% RSLogix 500 project PLC_TO_TURTLEBOT3.RSS, saved by version 12.00.00.00 %
PROJECT "ML1400"    % processor: MicroLogix 1400 %

PROGRAM FILES
  LAD 2   4 rungs
  LAD 3 "HMI"  5 rungs  % HMI Routine %
  LAD 4 "TELEOP"  7 rungs  % Modbus Routine %
  LAD 5 "COMMAND"  8 rungs

DATA FILES
  O0 OUTPUT  6 elements
  I1 INPUT  8 elements
  S2 STATUS  66 elements
  B3 BINARY  32 elements
  T4 TIMER  1 elements
  C5 COUNTER  1 elements
  R6 CONTROL  1 elements
  N7 INTEGER  20 elements
  F8 FLOAT  10 elements
  N9 HOLD_REG  25 elements
  F10 DECIMALES  7 elements
  N11   6 elements

LADDER 2
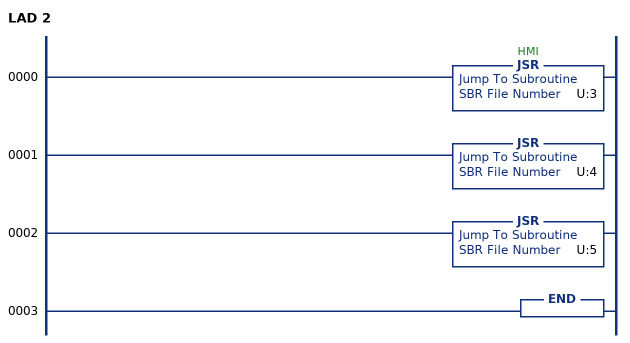
% Rung: 0 %
SOR JSR U:3 EOR
%   U:3  HMI %
% Rung: 1 %
SOR JSR U:4 EOR
% Rung: 2 %
SOR JSR U:5 EOR
% Rung: 3 %
SOR END EOR

LADDER 3 "HMI"    % HMI Routine %
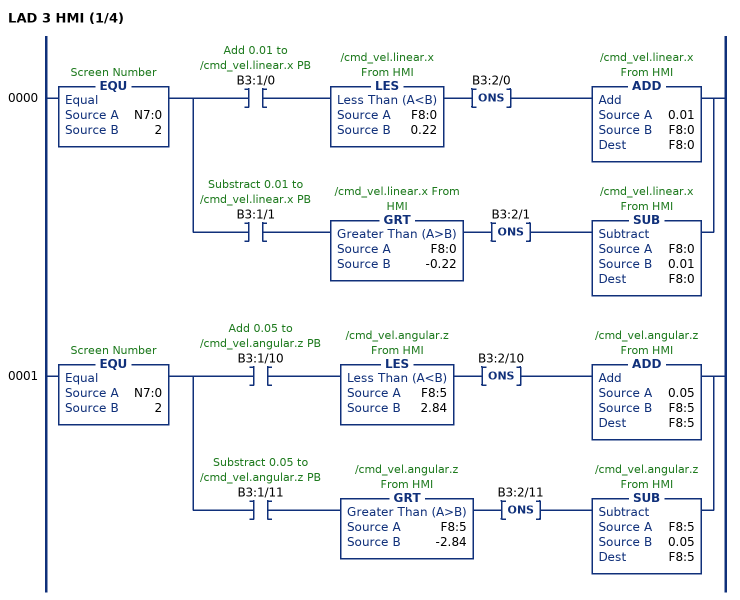
% Rung: 0 %
SOR EQU N7:0 2 BST XIC B3:1/0 LES F8:0 0.22 ONS B3:2/0 ADD 0.01 F8:0 F8:0 NXB XIC B3:1/1 GRT F8:0 -0.22 ONS B3:2/1 SUB F8:0 0.01 F8:0 BND EOR
%   N7:0  "Screen Number" %
%   B3:1/0  "Add 0.01 to /cmd_vel.linear.x PB" %
%   F8:0  "/cmd_vel.linear.x From HMI" %
%   B3:1/1  "Substract 0.01 to /cmd_vel.linear.x PB" %
% Rung: 1 %
SOR EQU N7:0 2 BST XIC B3:1/10 LES F8:5 2.84 ONS B3:2/10 ADD 0.05 F8:5 F8:5 NXB XIC B3:1/11 GRT F8:5 -2.84 ONS B3:2/11 SUB F8:5 0.05 F8:5 BND EOR
%   N7:0  "Screen Number" %
%   B3:1/10  "Add 0.05 to /cmd_vel.angular.z PB" %
%   F8:5  "/cmd_vel.angular.z From HMI" %
%   B3:1/11  "Substract 0.05 to /cmd_vel.angular.z PB" %

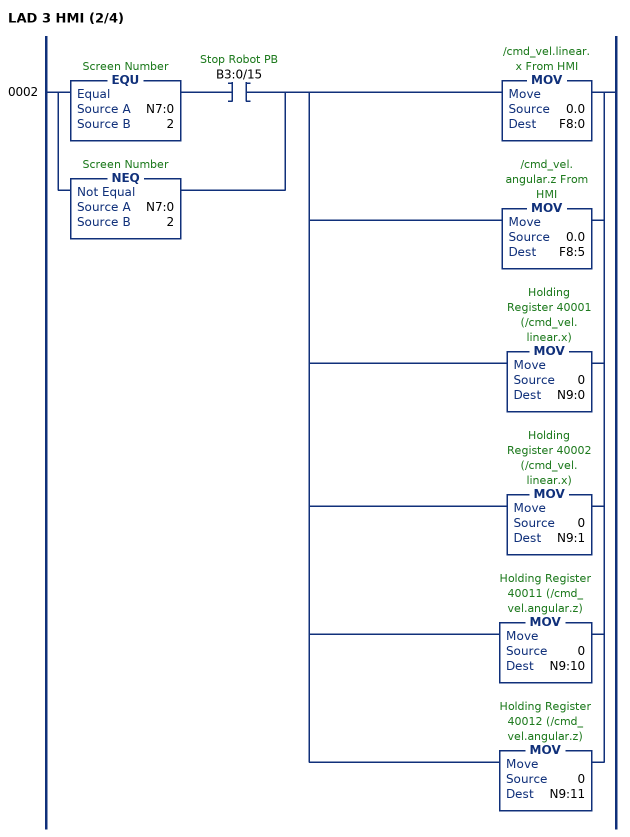
% Rung: 2 %
SOR BST EQU N7:0 2 XIC B3:0/15 NXB NEQ N7:0 2 BND BST MOV 0.0 F8:0 NXB MOV 0.0 F8:5 NXB MOV 0 N9:0 NXB MOV 0 N9:1 NXB MOV 0 N9:10 NXB MOV 0 N9:11 BND EOR
%   N7:0  "Screen Number" %
%   B3:0/15  "Stop Robot PB" %
%   F8:0  "/cmd_vel.linear.x From HMI" %
%   F8:5  "/cmd_vel.angular.z From HMI" %
%   N9:0  "Holding Register 40001 (/cmd_vel.linear.x)" %
%   N9:1  "Holding Register 40002 (/cmd_vel.linear.x)" %
%   N9:10  "Holding Register 40011 (/cmd_vel.angular.z)" %
%   N9:11  "Holding Register 40012 (/cmd_vel.angular.z)" %

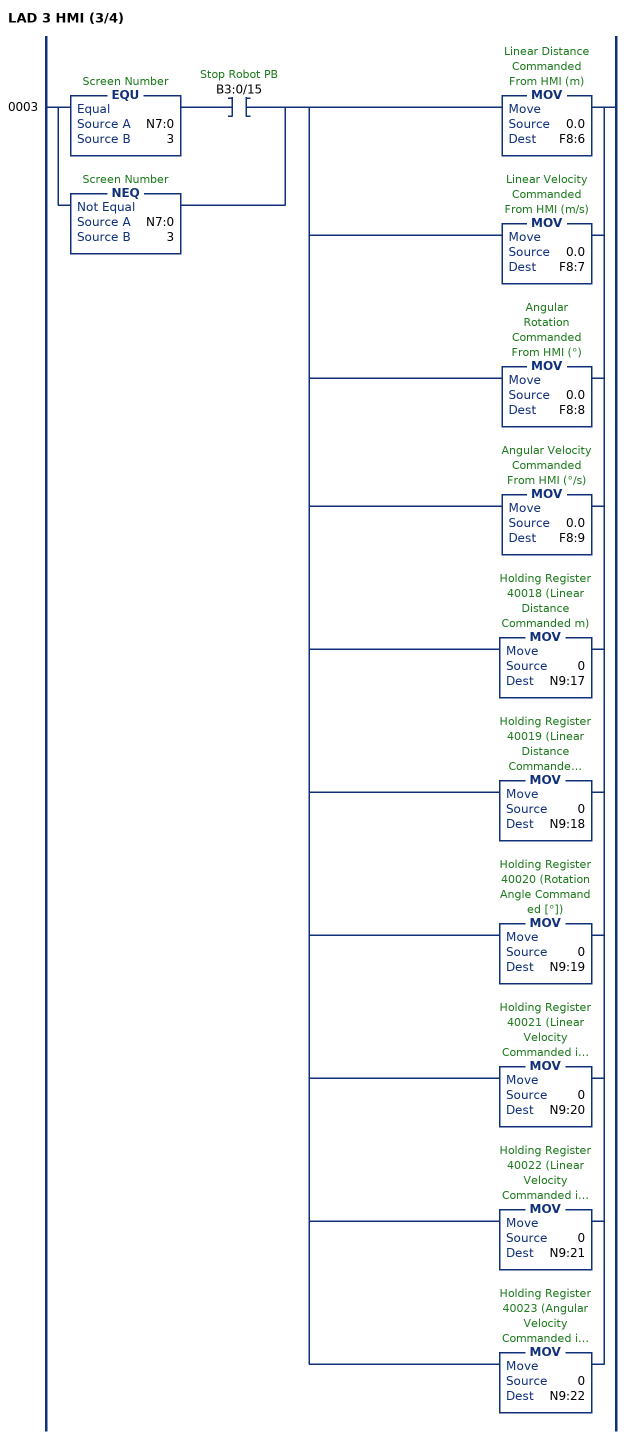
% Rung: 3 %
SOR BST EQU N7:0 3 XIC B3:0/15 NXB NEQ N7:0 3 BND BST MOV 0.0 F8:6 NXB MOV 0.0 F8:7 NXB MOV 0.0 F8:8 NXB MOV 0.0 F8:9 NXB MOV 0 N9:17 NXB MOV 0 N9:18 NXB MOV 0 N9:19 NXB MOV 0 N9:20 NXB MOV 0 N9:21 NXB MOV 0 N9:22 BND EOR
%   N7:0  "Screen Number" %
%   B3:0/15  "Stop Robot PB" %
%   F8:6  "Linear Distance Commanded From HMI (m)" %
%   F8:7  "Linear Velocity Commanded From HMI (m/s)" %
%   F8:8  "Angular Rotation Commanded From HMI (°)" %
%   F8:9  "Angular Velocity Commanded From HMI (°/s)" %
%   N9:17  "Holding Register 40018 (Linear Distance Commanded m)" %
%   N9:18  "Holding Register 40019 (Linear Distance Commanded cm)" %
%   N9:19  "Holding Register 40020 (Rotation Angle Commanded [°])" %
%   N9:20  "Holding Register 40021 (Linear Velocity Commanded in X axis [m])" %
%   N9:21  "Holding Register 40022 (Linear Velocity Commanded in X axis [cm])" %
%   N9:22  "Holding Register 40023 (Angular Velocity Commanded in Z axis [°/s])" %

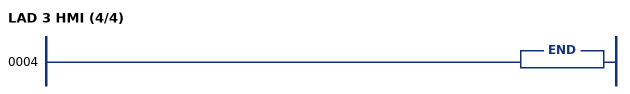
% Rung: 4 %
SOR END EOR

LADDER 4 "TELEOP"    % Modbus Routine %
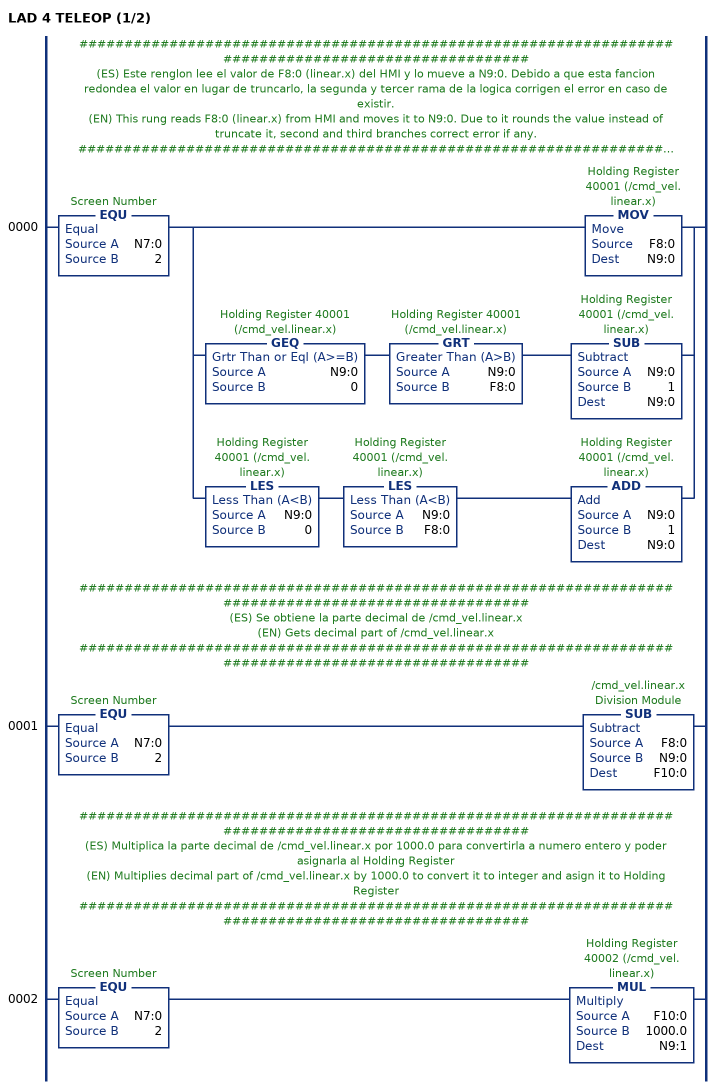
% Rung: 0 %
% ####################################################################################################
% 
% (ES) Este renglon lee el valor de F8:0 (linear.x) del HMI y lo mueve a N9:0. Debido a que esta fancion redondea el valor en lugar de truncarlo, la segunda y tercer rama de la logica corrigen el error en caso de existir.
% (EN) This rung reads F8:0 (linear.x) from HMI and moves it to N9:0. Due to it rounds the value instead of truncate it, second and third branches correct error if any.
% 
% #################################################################################################### %
SOR EQU N7:0 2 BST MOV F8:0 N9:0 NXB GEQ N9:0 0 GRT N9:0 F8:0 SUB N9:0 1 N9:0 NXB LES N9:0 0 LES N9:0 F8:0 ADD N9:0 1 N9:0 BND EOR
%   N7:0  "Screen Number" %
%   F8:0  "/cmd_vel.linear.x From HMI" %
%   N9:0  "Holding Register 40001 (/cmd_vel.linear.x)" %
% Rung: 1 %
% ####################################################################################################
% 
% (ES) Se obtiene la parte decimal de /cmd_vel.linear.x
% (EN) Gets decimal part of /cmd_vel.linear.x
% 
% #################################################################################################### %
SOR EQU N7:0 2 SUB F8:0 N9:0 F10:0 EOR
%   N7:0  "Screen Number" %
%   F8:0  "/cmd_vel.linear.x From HMI" %
%   N9:0  "Holding Register 40001 (/cmd_vel.linear.x)" %
%   F10:0  "/cmd_vel.linear.x Division Module" %
% Rung: 2 %
% ####################################################################################################
% 
% (ES) Multiplica la parte decimal de /cmd_vel.linear.x por 1000.0 para convertirla a numero entero y poder asignarla al Holding Register
% (EN) Multiplies decimal part of /cmd_vel.linear.x by 1000.0 to convert it to integer and asign it to Holding Register
% 
% #################################################################################################### %
SOR EQU N7:0 2 MUL F10:0 1000.0 N9:1 EOR
%   N7:0  "Screen Number" %
%   F10:0  "/cmd_vel.linear.x Division Module" %
%   N9:1  "Holding Register 40002 (/cmd_vel.linear.x)" %

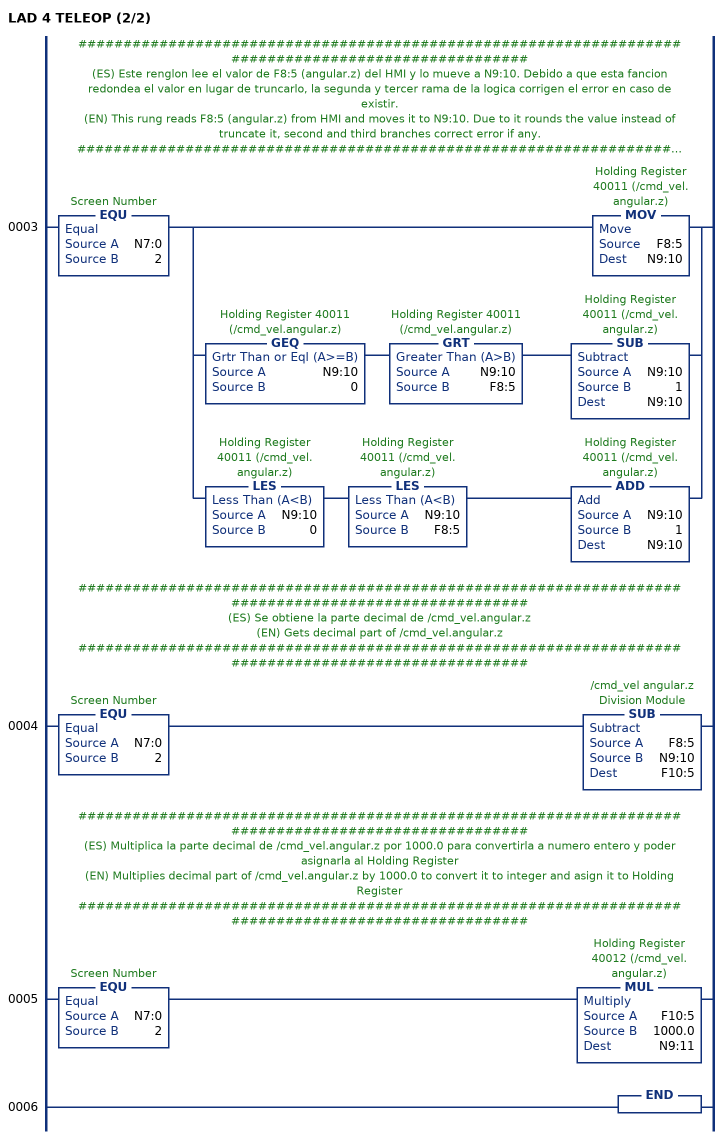
% Rung: 3 %
% ####################################################################################################
% 
% (ES) Este renglon lee el valor de F8:5 (angular.z) del HMI y lo mueve a N9:10. Debido a que esta fancion redondea el valor en lugar de truncarlo, la segunda y tercer rama de la logica corrigen el error en caso de existir.
% (EN) This rung reads F8:5 (angular.z) from HMI and moves it to N9:10. Due to it rounds the value instead of truncate it, second and third branches correct error if any.
% 
% #################################################################################################### %
SOR EQU N7:0 2 BST MOV F8:5 N9:10 NXB GEQ N9:10 0 GRT N9:10 F8:5 SUB N9:10 1 N9:10 NXB LES N9:10 0 LES N9:10 F8:5 ADD N9:10 1 N9:10 BND EOR
%   N7:0  "Screen Number" %
%   F8:5  "/cmd_vel.angular.z From HMI" %
%   N9:10  "Holding Register 40011 (/cmd_vel.angular.z)" %
% Rung: 4 %
% ####################################################################################################
% 
% (ES) Se obtiene la parte decimal de /cmd_vel.angular.z
% (EN) Gets decimal part of /cmd_vel.angular.z
% 
% #################################################################################################### %
SOR EQU N7:0 2 SUB F8:5 N9:10 F10:5 EOR
%   N7:0  "Screen Number" %
%   F8:5  "/cmd_vel.angular.z From HMI" %
%   N9:10  "Holding Register 40011 (/cmd_vel.angular.z)" %
%   F10:5  "/cmd_vel angular.z Division Module" %
% Rung: 5 %
% ####################################################################################################
% 
% (ES) Multiplica la parte decimal de /cmd_vel.angular.z por 1000.0 para convertirla a numero entero y poder asignarla al Holding Register
% (EN) Multiplies decimal part of /cmd_vel.angular.z by 1000.0 to convert it to integer and asign it to Holding Register
% 
% #################################################################################################### %
SOR EQU N7:0 2 MUL F10:5 1000.0 N9:11 EOR
%   N7:0  "Screen Number" %
%   F10:5  "/cmd_vel angular.z Division Module" %
%   N9:11  "Holding Register 40012 (/cmd_vel.angular.z)" %
% Rung: 6 %
SOR END EOR

LADDER 5 "COMMAND"
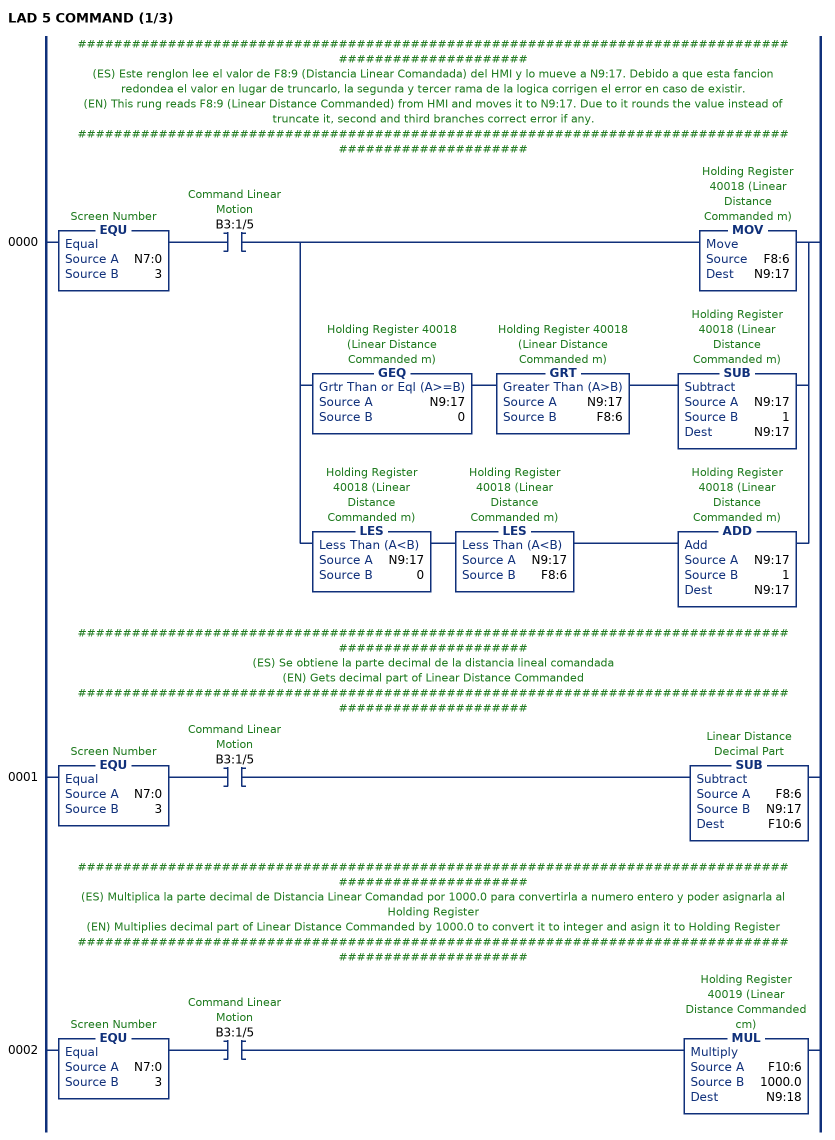
% Rung: 0 %
% ####################################################################################################
% 
% (ES) Este renglon lee el valor de F8:9 (Distancia Linear Comandada) del HMI y lo mueve a N9:17. Debido a que esta fancion redondea el valor en lugar de truncarlo, la segunda y tercer rama de la logica corrigen el error en caso de existir.
% (EN) This rung reads F8:9 (Linear Distance Commanded) from HMI and moves it to N9:17. Due to it rounds the value instead of truncate it, second and third branches correct error if any.
% 
% #################################################################################################### %
SOR EQU N7:0 3 XIC B3:1/5 BST MOV F8:6 N9:17 NXB GEQ N9:17 0 GRT N9:17 F8:6 SUB N9:17 1 N9:17 NXB LES N9:17 0 LES N9:17 F8:6 ADD N9:17 1 N9:17 BND EOR
%   N7:0  "Screen Number" %
%   B3:1/5  "Command Linear Motion" %
%   F8:6  "Linear Distance Commanded From HMI (m)" %
%   N9:17  "Holding Register 40018 (Linear Distance Commanded m)" %
% Rung: 1 %
% ####################################################################################################
% 
% (ES) Se obtiene la parte decimal de la distancia lineal comandada
% (EN) Gets decimal part of Linear Distance Commanded
% 
% #################################################################################################### %
SOR EQU N7:0 3 XIC B3:1/5 SUB F8:6 N9:17 F10:6 EOR
%   N7:0  "Screen Number" %
%   B3:1/5  "Command Linear Motion" %
%   F8:6  "Linear Distance Commanded From HMI (m)" %
%   N9:17  "Holding Register 40018 (Linear Distance Commanded m)" %
%   F10:6  "Linear Distance Decimal Part" %
% Rung: 2 %
% ####################################################################################################
% 
% (ES) Multiplica la parte decimal de Distancia Linear Comandad por 1000.0 para convertirla a numero entero y poder asignarla al Holding Register
% (EN) Multiplies decimal part of Linear Distance Commanded by 1000.0 to convert it to integer and asign it to Holding Register
% 
% #################################################################################################### %
SOR EQU N7:0 3 XIC B3:1/5 MUL F10:6 1000.0 N9:18 EOR
%   N7:0  "Screen Number" %
%   B3:1/5  "Command Linear Motion" %
%   F10:6  "Linear Distance Decimal Part" %
%   N9:18  "Holding Register 40019 (Linear Distance Commanded cm)" %

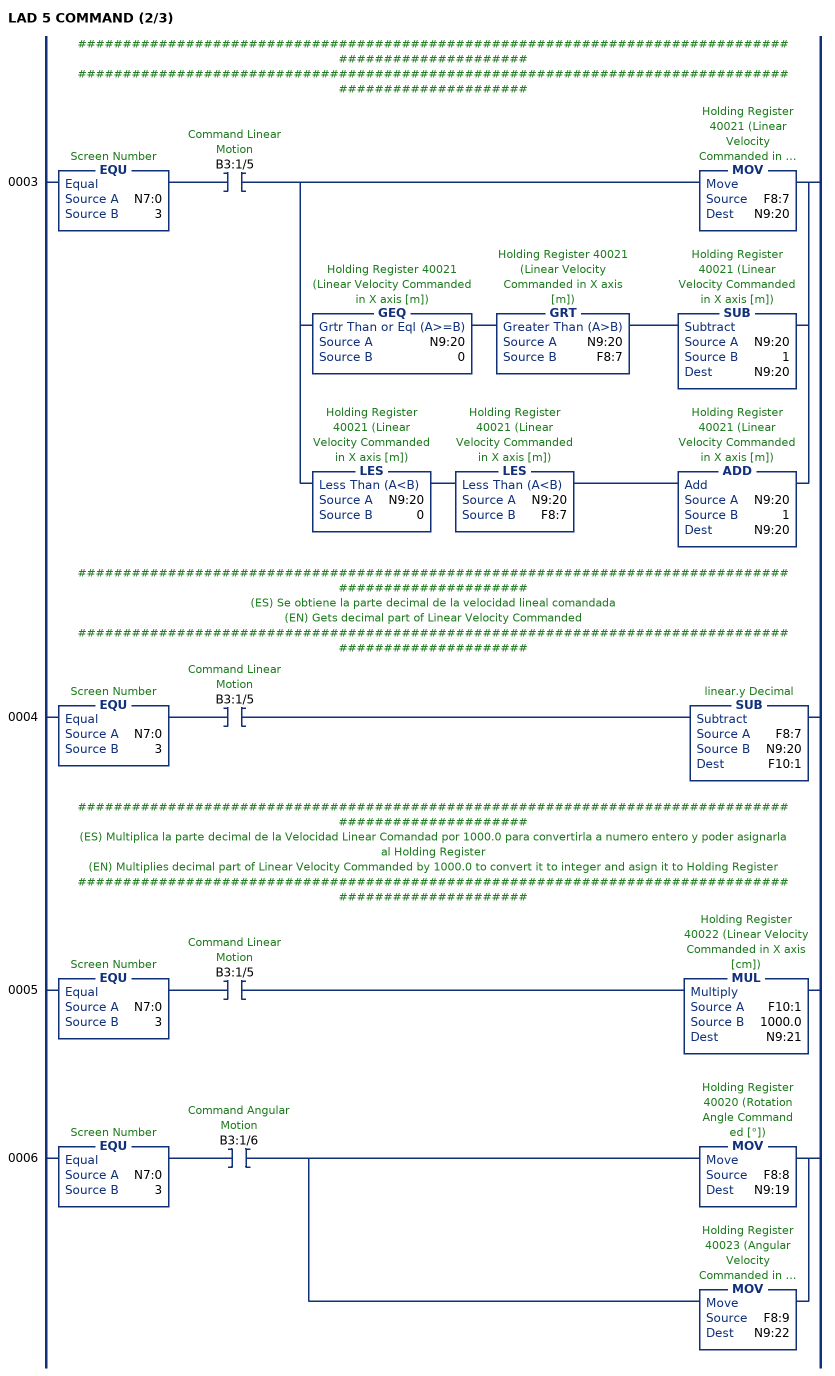
% Rung: 3 %
% ####################################################################################################
% 
% 
% 
% #################################################################################################### %
SOR EQU N7:0 3 XIC B3:1/5 BST MOV F8:7 N9:20 NXB GEQ N9:20 0 GRT N9:20 F8:7 SUB N9:20 1 N9:20 NXB LES N9:20 0 LES N9:20 F8:7 ADD N9:20 1 N9:20 BND EOR
%   N7:0  "Screen Number" %
%   B3:1/5  "Command Linear Motion" %
%   F8:7  "Linear Velocity Commanded From HMI (m/s)" %
%   N9:20  "Holding Register 40021 (Linear Velocity Commanded in X axis [m])" %
% Rung: 4 %
% ####################################################################################################
% 
% (ES) Se obtiene la parte decimal de la velocidad lineal comandada
% (EN) Gets decimal part of Linear Velocity Commanded
% 
% #################################################################################################### %
SOR EQU N7:0 3 XIC B3:1/5 SUB F8:7 N9:20 F10:1 EOR
%   N7:0  "Screen Number" %
%   B3:1/5  "Command Linear Motion" %
%   F8:7  "Linear Velocity Commanded From HMI (m/s)" %
%   N9:20  "Holding Register 40021 (Linear Velocity Commanded in X axis [m])" %
%   F10:1  "linear.y Decimal" %
% Rung: 5 %
% ####################################################################################################
% 
% (ES) Multiplica la parte decimal de la Velocidad Linear Comandad por 1000.0 para convertirla a numero entero y poder asignarla al Holding Register
% (EN) Multiplies decimal part of Linear Velocity Commanded by 1000.0 to convert it to integer and asign it to Holding Register
% 
% #################################################################################################### %
SOR EQU N7:0 3 XIC B3:1/5 MUL F10:1 1000.0 N9:21 EOR
%   N7:0  "Screen Number" %
%   B3:1/5  "Command Linear Motion" %
%   F10:1  "linear.y Decimal" %
%   N9:21  "Holding Register 40022 (Linear Velocity Commanded in X axis [cm])" %
% Rung: 6 %
SOR EQU N7:0 3 XIC B3:1/6 BST MOV F8:8 N9:19 NXB MOV F8:9 N9:22 BND EOR
%   N7:0  "Screen Number" %
%   B3:1/6  "Command Angular Motion" %
%   F8:8  "Angular Rotation Commanded From HMI (°)" %
%   N9:19  "Holding Register 40020 (Rotation Angle Commanded [°])" %
%   F8:9  "Angular Velocity Commanded From HMI (°/s)" %
%   N9:22  "Holding Register 40023 (Angular Velocity Commanded in Z axis [°/s])" %

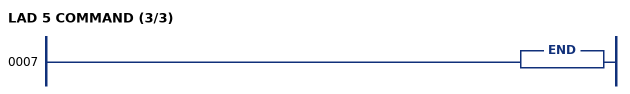
% Rung: 7 %
SOR END EOR

OTHER DOCUMENTED ADDRESSES
  B3:1/2  "Add 0.05 to /cmd_vel.angular.z PB"
  B3:1/3  "Substract 0.05 to /cmd_vel.angular.z PB"
  F8:1  "/cmd_vel.linear.y From HMI (Unused in TB3)"
  F8:2  "/cmd_vel.linear.z From HMI (Unused in TB3)"
  F8:3  "/cmd_vel.angular.x From HMI (Unused in TB3)"
  F8:4  "/cmd_vel.angular.y From HMI (Unused in TB3)"
  F10:2  "linear.z Decimal"
  F10:3  "angular.x Decimal"
  F10:4  "angular.y Decimal"
  N7:10  "Rotation Angle Commanded From HMI (Deg)"
  N9:2  "Holding Register 40003 (/cmd_vel.linear.y)"
  N9:3  "Holding Register 40004 (/cmd_vel.linear.y)"
  N9:4  "Holding Register 40005 (/cmd_vel.linear.z)"
  N9:5  "Holding Register 40006 (/cmd_vel.linear.z)"
  N9:6  "Holding Register 40007 (/cmd_vel.angular.x)"
  N9:7  "Holding Register 40008 (/cmd_vel.angular.x)"
  N9:8  "Holding Register 40009 (/cmd_vel.angular.y)"
  N9:9  "Holding Register 40010 (/cmd_vel.angular.y)"
  N9:12  "Holding Register 40013 (Spare)"
  N9:13  "Holding Register 40014 (Spare)"
  N9:14  "Holding Register 40015 (Spare)"
  N9:15  "Holding Register 40016 (Spare)"
  N9:16  "Holding Register 40017 (Spare)"

DATA TABLE (non-zero values as saved)
DATA N7
% N7:0 % 2 0 0 0 0 0 0 0 0 0
DATA F10
% F10:0 % 0 0.18 0 0 0
% F10:5 % 0 0.4
DATA N11
% N11:0 % 5 240 0 0 0 0
